Fanuc KAREL source: compact_preamble.KL

PROGRAM KB00132
%NOLOCKGROUP
VAR
P1 : STRING[80];P2:INTEGER;P3:INTEGER
BEGIN
P1='A'
P2=1
P3=1
POP_KEY_RD(P1,P2,P3)
END KB00132
